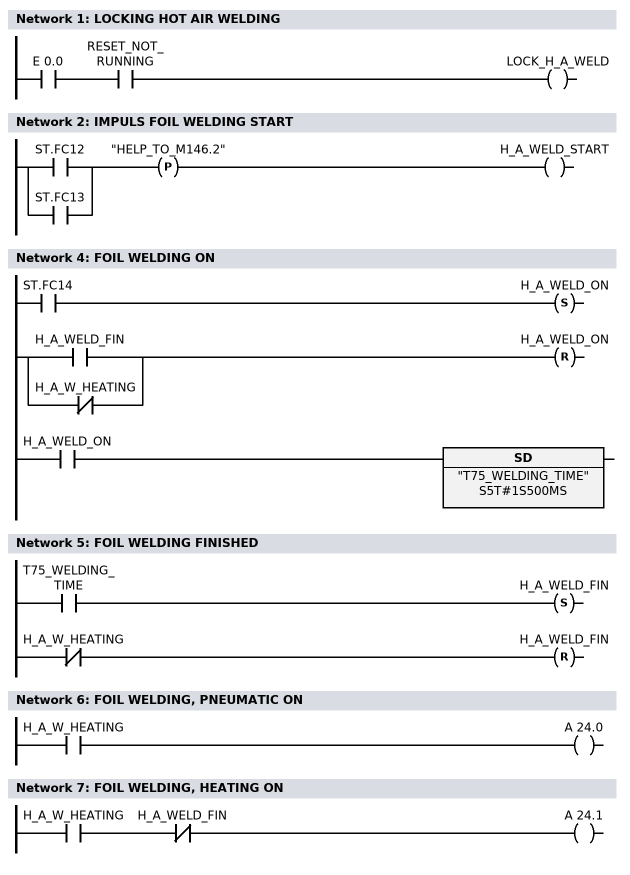
[picture p48: HOT_AIR_WELDING networks 1-7]
NETWORK
TITLE = LOCKING HOT AIR WELDING
//Verriegelung Folie ansiegeln
      A     "E 0.0";
      A     "RESET_NOT_RUNNING";
      =     "LOCK_H_A_WELD";
NETWORK
TITLE = IMPULS FOIL WELDING START 
//Impuls Folie ansiegeln ein
      A(;
      O     "ST.FC12";
      O     "ST.FC13";
      );
      FP    "HELP_TO_M146.2";
      =     "H_A_WELD_START";
NETWORK
TITLE = FOIL WELDING HEATING 
//Folie ansiegeln ein
      A(;
      A     "H_A_WELD_START";
      S     "H_A_W_HEATING";
      A(;
      ON    "LOCK_H_A_WELD";
      O     "T74_HEATING_TIME";
      );
      R     "H_A_W_HEATING";
      A     "H_A_W_HEATING";
      );
      A     "H_A_WELD_FIN";
      L     S5T#15S;
      SD    "T74_HEATING_TIME";
NETWORK
TITLE = FOIL WELDING ON
//Folie ansiegeln aktiv
      A     "ST.FC14";
      S     "H_A_WELD_ON";
      A(;
      O     "H_A_WELD_FIN";
      ON    "H_A_W_HEATING";
      );
      R     "H_A_WELD_ON";
      A     "H_A_WELD_ON";
      L     S5T#1S500MS;
      SD    "T75_WELDING_TIME";
NETWORK
TITLE = FOIL WELDING FINISHED
//Folie ansiegeln fertig
      A     "T75_WELDING_TIME";
      S     "H_A_WELD_FIN";
      AN    "H_A_W_HEATING";
      R     "H_A_WELD_FIN";
      NOP   0;
NETWORK
TITLE = FOIL WELDING, PNEUMATIC ON
//Folie ansiegeln Luft ein
      A     "H_A_W_HEATING";
      =     "A 24.0";
NETWORK
TITLE = FOIL WELDING, HEATING ON
//Folie ansiegeln Heizung ein
      A     "H_A_W_HEATING";
      AN    "H_A_WELD_FIN";
      =     "A 24.1";
END_FUNCTION

FUNCTION "WELDING" : VOID	// FC 29
TITLE = FILM WELDING, OPTION
AUTHOR : LKA
NAME : WELDING
VERSION : 0.1
BEGIN
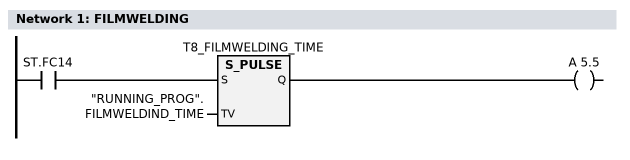
NETWORK
TITLE = FILMWELDING
      A     "ST.FC14";
      L     "RUNNING_PROG".FILMWELDIND_TIME;
      SP    "T8_FILMWELDING_TIME";
      NOP   0;
      NOP   0;
      NOP   0;
      A     "T8_FILMWELDING_TIME";
      =     "A 5.5";
END_FUNCTION

FUNCTION "TURNTABLE_COUNTERS" : VOID	// FC 32
TITLE = TURNTABLE COUNTERS AND TIMERS
//HELP FUNCTION TO PROGRAM, COMMON COUNTERS USED IN WRAPPING PROGRAMMS
AUTHOR : LKA
NAME : FROM_TOP
VERSION : 0.1
BEGIN
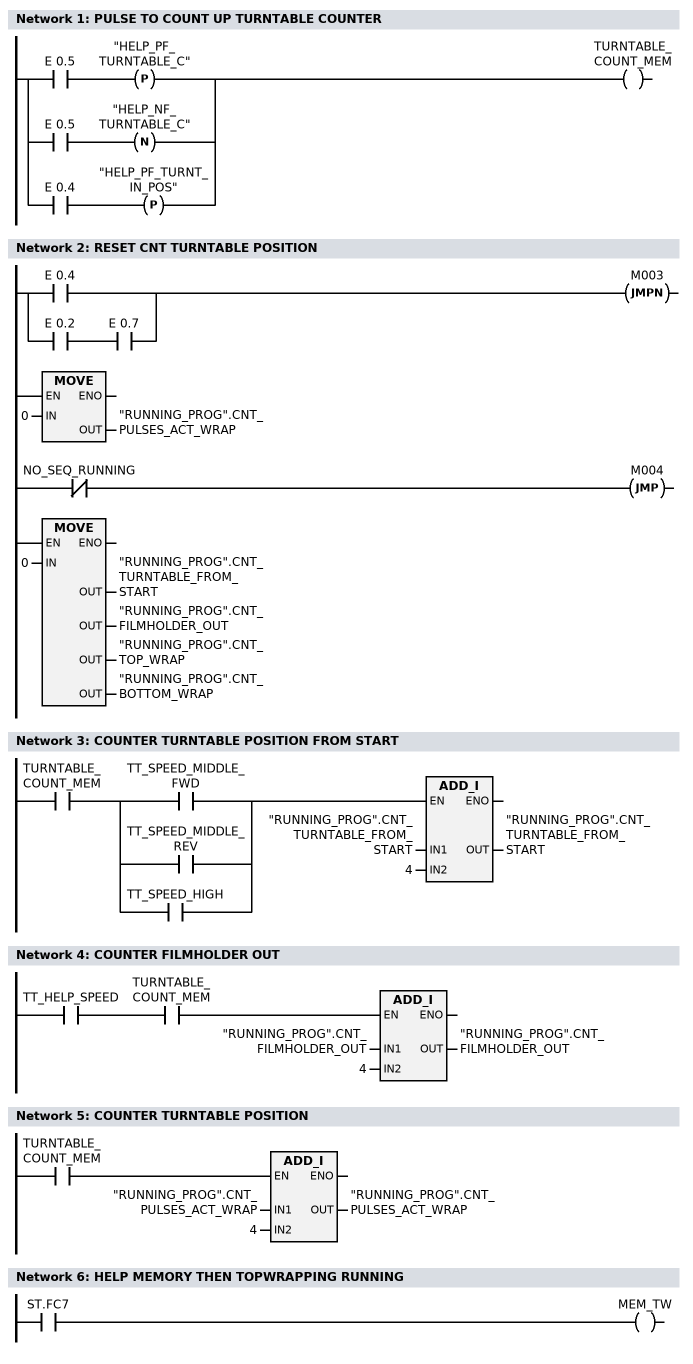
NETWORK
TITLE = PULSE TO COUNT UP TURNTABLE COUNTER
      A     "E 0.5";
      FP    "HELP_PF_TURNTABLE_C";
      O(;
      A     "E 0.5";
      FN    "HELP_NF_TURNTABLE_C";
      );
      O(;
      A     "E 0.4";
      FP    "HELP_PF_TURNT_IN_POS";
      );
      =     "TURNTABLE_COUNT_MEM";
NETWORK
TITLE = RESET CNT TURNTABLE POSITION
//RESETA BORD POSITIONS RÄKNARE
      O     "E 0.4";
      O;
      A     "E 0.2";
      A     "E 0.7";
      JCN   M003;
      L     0;
      T     "RUNNING_PROG".CNT_PULSES_ACT_WRAP;
M003: NOP   0;
      AN    "NO_SEQ_RUNNING";	// OM INTE NÅGON CYKEL KÖRS
      JC    M004;
      L     0;
      T     "RUNNING_PROG".CNT_TURNTABLE_FROM_START;
      T     "RUNNING_PROG".CNT_FILMHOLDER_OUT;
      T     "RUNNING_PROG".CNT_TOP_WRAP;
      T     "RUNNING_PROG".CNT_BOTTOM_WRAP;
M004: NOP   0;
NETWORK
TITLE = COUNTER TURNTABLE POSITION FROM START
//RÄKNARE BORD POSITION
      A     "TURNTABLE_COUNT_MEM";
      A(;
      O     "TT_SPEED_MIDDLE_FWD";
      O     "TT_SPEED_MIDDLE_REV";
      O     "TT_SPEED_HIGH";
      );
      JNB   _008;
      L     "RUNNING_PROG".CNT_TURNTABLE_FROM_START;
      L     4;
      +I;
      T     "RUNNING_PROG".CNT_TURNTABLE_FROM_START;
_008: NOP   0;
NETWORK
TITLE = COUNTER FILMHOLDER OUT
//RÄKNARE FILMHÅLLARARM UT, samt när byte till hög fart skall ske!
      A     "TT_HELP_SPEED";
      A     "TURNTABLE_COUNT_MEM";
      JNB   _00b;
      L     "RUNNING_PROG".CNT_FILMHOLDER_OUT;
      L     4;
      +I;
      T     "RUNNING_PROG".CNT_FILMHOLDER_OUT;
_00b: NOP   0;
NETWORK
TITLE = COUNTER TURNTABLE POSITION
//RÄKNARE BORD POSITION
      A     "TURNTABLE_COUNT_MEM";
      JNB   _010;
      L     "RUNNING_PROG".CNT_PULSES_ACT_WRAP;
      L     4;
      +I;
      T     "RUNNING_PROG".CNT_PULSES_ACT_WRAP;
_010: NOP   0;
NETWORK
TITLE = HELP MEMORY THEN TOPWRAPPING RUNNING
//HJÄLP MINNE FÖR NÄR TOPP VARV KÖRS
      A     "ST.FC7";
      =     "MEM_TW";
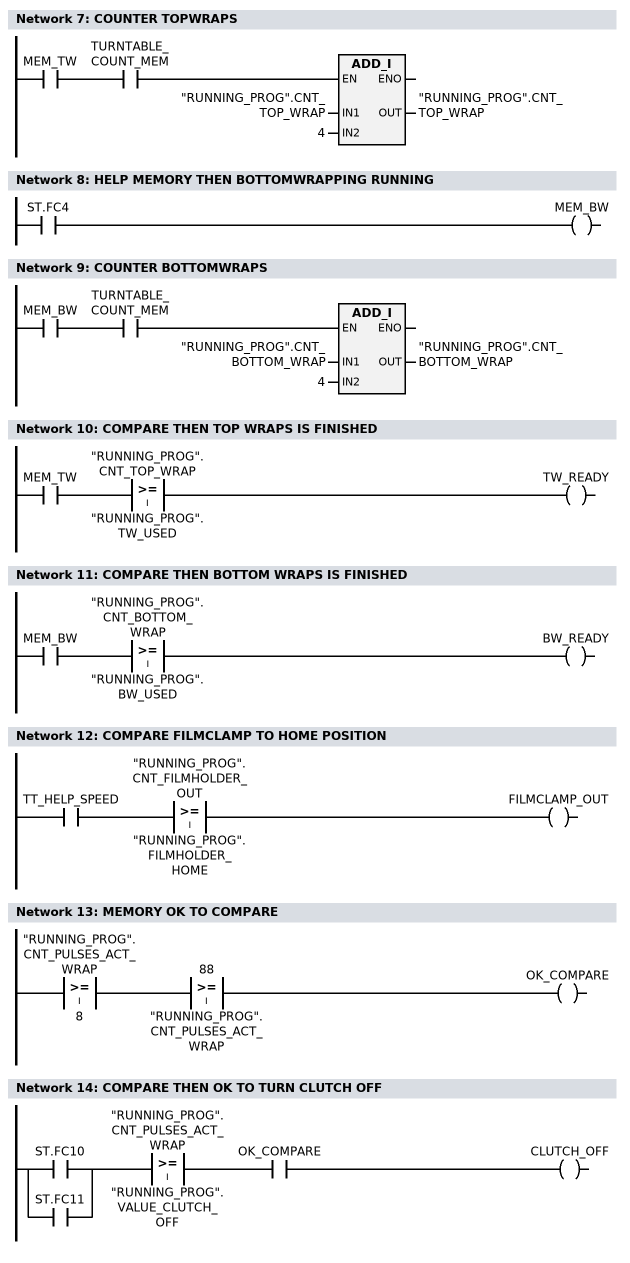
NETWORK
TITLE = COUNTER TOPWRAPS
//RÄKNARE TOPP VARV
      A     "MEM_TW";
      A     "TURNTABLE_COUNT_MEM";
      JNB   _011;
      L     "RUNNING_PROG".CNT_TOP_WRAP;
      L     4;
      +I;
      T     "RUNNING_PROG".CNT_TOP_WRAP;
_011: NOP   0;
NETWORK
TITLE = HELP MEMORY THEN BOTTOMWRAPPING RUNNING
//HJÄLP MINNE FÖR NÄR BOTTEN VARV KÖRS
      A     "ST.FC4";
      =     "MEM_BW";
NETWORK
TITLE = COUNTER BOTTOMWRAPS
//RÄKNARE BOTTEN VARV
      A     "MEM_BW";
      A     "TURNTABLE_COUNT_MEM";
      JNB   _012;
      L     "RUNNING_PROG".CNT_BOTTOM_WRAP;
      L     4;
      +I;
      T     "RUNNING_PROG".CNT_BOTTOM_WRAP;
_012: NOP   0;
NETWORK
TITLE = COMPARE THEN TOP WRAPS IS FINISHED
//HJÄLP MINNE TILL NÄR TOPPVARV ÄR KLARA
      A     "MEM_TW";
      A(;
      L     "RUNNING_PROG".CNT_TOP_WRAP;
      L     "RUNNING_PROG".TW_USED;
      >=I;
      );
      =     "TW_READY";
NETWORK
TITLE = COMPARE THEN BOTTOM WRAPS IS FINISHED
//HJÄLP MINNE TILL NÄR BOTTENVARV ÄR KLARA
//BYTT DB12.DBW80 MOT 78??!!!!
      A     "MEM_BW";
      A(;
      L     "RUNNING_PROG".CNT_BOTTOM_WRAP;
      L     "RUNNING_PROG".BW_USED;
      >=I;
      );
      =     "BW_READY";
NETWORK
TITLE = COMPARE FILMCLAMP TO HOME POSITION
//HJÄLP MINNE TILL NÄR FILMHÅLLARARM SKALL UT
//
      A     "TT_HELP_SPEED";
      A(;
      L     "RUNNING_PROG".CNT_FILMHOLDER_OUT;
      L     "RUNNING_PROG".FILMHOLDER_HOME;
      >=I;
      );
      =     "FILMCLAMP_OUT";
NETWORK
TITLE = MEMORY OK TO COMPARE
      A(;
      L     "RUNNING_PROG".CNT_PULSES_ACT_WRAP;
      L     8;
      >=I;
      );
      A(;
      L     88;
      L     "RUNNING_PROG".CNT_PULSES_ACT_WRAP;
      >=I;
      );
      =     "OK_COMPARE";
NETWORK
TITLE = COMPARE THEN OK TO TURN CLUTCH OFF
      A(;
      O     "ST.FC10";
      O     "ST.FC11";
      );
      A(;
      L     "RUNNING_PROG".CNT_PULSES_ACT_WRAP;
      L     "RUNNING_PROG".VALUE_CLUTCH_OFF;
      >=I;
      );
      A     "OK_COMPARE";
      =     "CLUTCH_OFF";
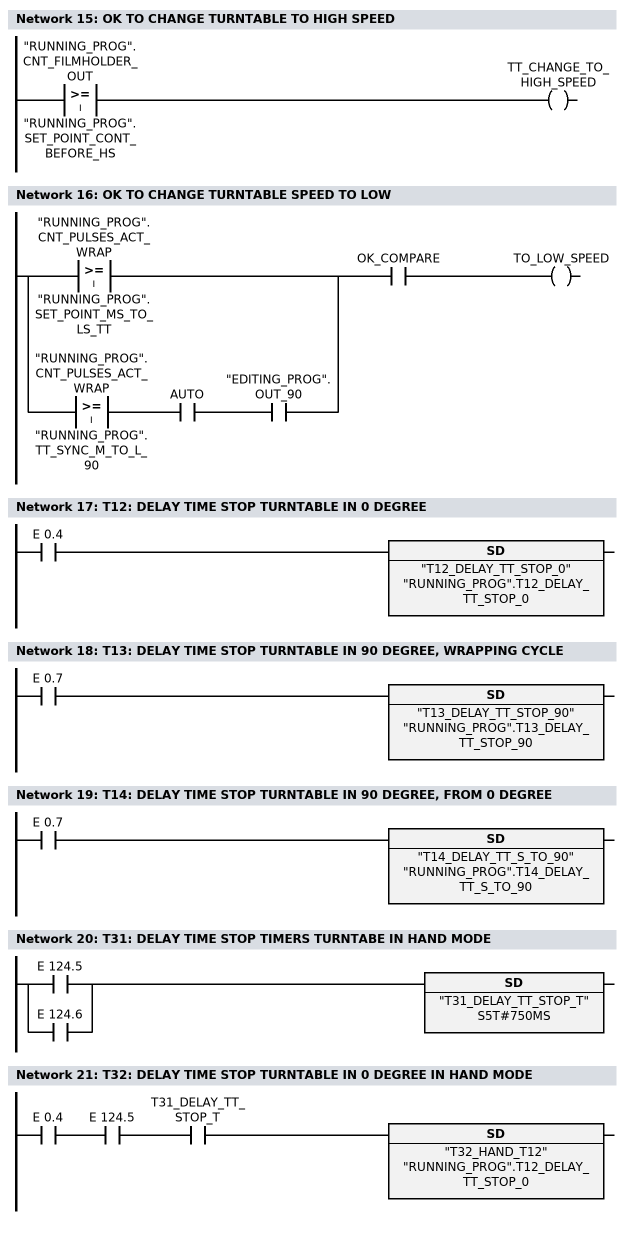
NETWORK
TITLE = OK TO CHANGE TURNTABLE TO HIGH SPEED
//HJÄLP MINNE TILL NÄR BORDET ÄR I POSITION SÅ DET ÄR OK ATT ÖKA TILL HÖGFART
      L     "RUNNING_PROG".CNT_FILMHOLDER_OUT;
      L     "RUNNING_PROG".SET_POINT_CONT_BEFORE_HS;
      >=I;
      =     "TT_CHANGE_TO_HIGH_SPEED";
NETWORK
TITLE = OK TO CHANGE TURNTABLE SPEED TO LOW
      A(;
      O(;
      L     "RUNNING_PROG".CNT_PULSES_ACT_WRAP;
      L     "RUNNING_PROG".SET_POINT_MS_TO_LS_TT;
      >=I;
      );
      O;
      A(;
      L     "RUNNING_PROG".CNT_PULSES_ACT_WRAP;
      L     "RUNNING_PROG".TT_SYNC_M_TO_L_90;
      >=I;
      );
      A     "AUTO";
      A     "EDITING_PROG".OUT_90;
      );
      A     "OK_COMPARE";
      =     "TO_LOW_SPEED";
NETWORK
TITLE = T12: DELAY TIME STOP TURNTABLE IN 0 DEGREE
      A     "E 0.4";
      L     "RUNNING_PROG".T12_DELAY_TT_STOP_0;
      SD    "T12_DELAY_TT_STOP_0";
NETWORK
TITLE = T13: DELAY TIME STOP TURNTABLE IN 90 DEGREE, WRAPPING CYCLE
      A     "E 0.7";
      L     "RUNNING_PROG".T13_DELAY_TT_STOP_90;
      SD    "T13_DELAY_TT_STOP_90";
NETWORK
TITLE = T14: DELAY TIME STOP TURNTABLE IN 90 DEGREE, FROM 0 DEGREE
      A     "E 0.7";
      L     "RUNNING_PROG".T14_DELAY_TT_S_TO_90;
      SD    "T14_DELAY_TT_S_TO_90";
NETWORK
TITLE = T31: DELAY TIME STOP TIMERS TURNTABE IN HAND MODE
      O     "E 124.5";
      O     "E 124.6";
      L     S5T#750MS;
      SD    "T31_DELAY_TT_STOP_T";
NETWORK
TITLE = T32: DELAY TIME STOP TURNTABLE IN 0 DEGREE IN HAND MODE
      A     "E 0.4";
      A     "E 124.5";
      A     "T31_DELAY_TT_STOP_T";
      L     "RUNNING_PROG".T12_DELAY_TT_STOP_0;
      SD    "T32_HAND_T12";
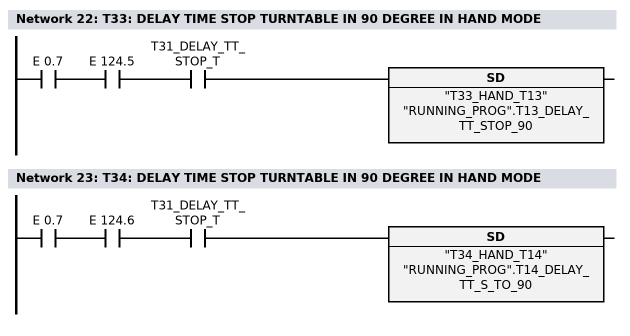
NETWORK
TITLE = T33: DELAY TIME STOP TURNTABLE IN 90 DEGREE IN HAND MODE
      A     "E 0.7";
      A     "E 124.5";
      A     "T31_DELAY_TT_STOP_T";
      L     "RUNNING_PROG".T13_DELAY_TT_STOP_90;
      SD    "T33_HAND_T13";
NETWORK
TITLE = T34: DELAY TIME STOP TURNTABLE IN 90 DEGREE IN HAND MODE
      A     "E 0.7";
      A     "E 124.6";
      A     "T31_DELAY_TT_STOP_T";
      L     "RUNNING_PROG".T14_DELAY_TT_S_TO_90;
      SD    "T34_HAND_T14";
END_FUNCTION

FUNCTION "CARRIAGE_COUNTERS" : VOID	// FC 33
TITLE = CARRIAGE COUNTERS
//HELP FUNCTION TO PROGRAM, COMMON COUNTERS USED IN WRAPPING PROGRAMMS
AUTHOR : LKA
NAME : FROM_TOP
VERSION : 0.1
BEGIN
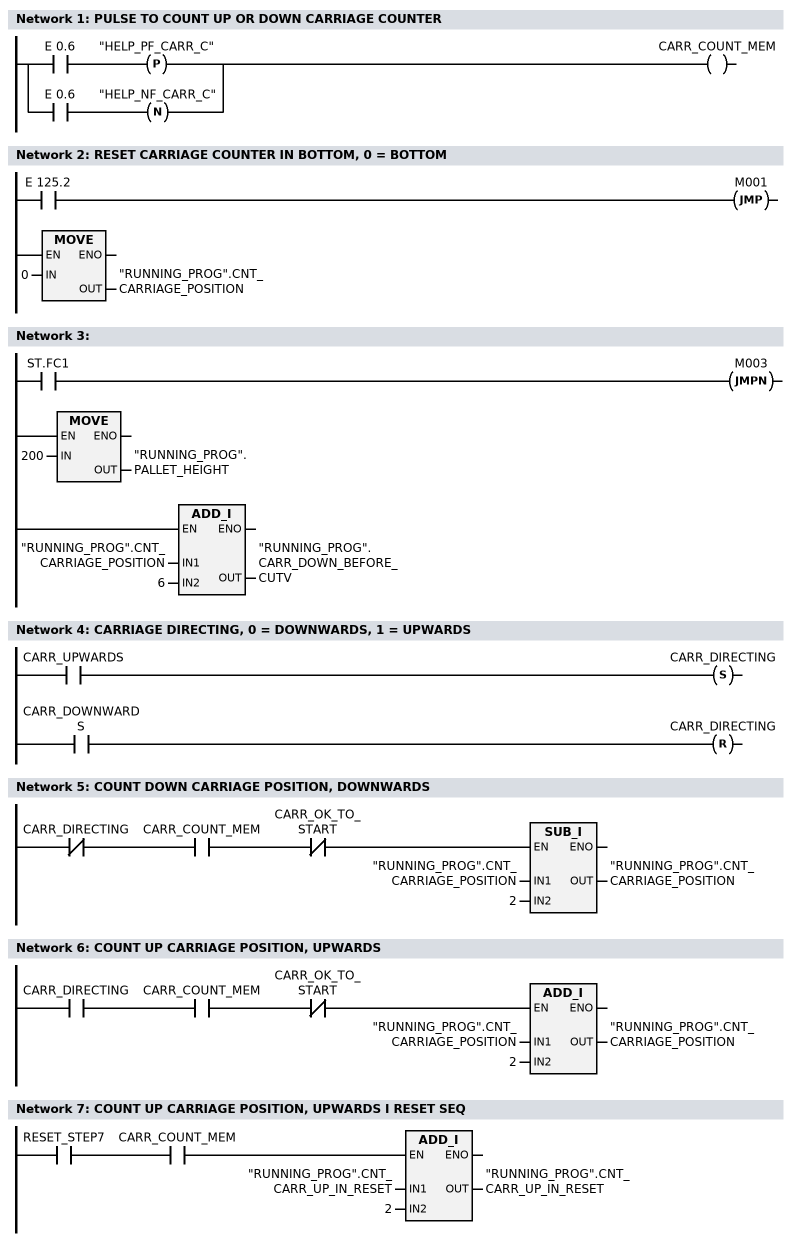
NETWORK
TITLE = PULSE TO COUNT UP OR DOWN CARRIAGE COUNTER
      A     "E 0.6";
      FP    "HELP_PF_CARR_C";
      O(;
      A     "E 0.6";
      FN    "HELP_NF_CARR_C";
      );
      =     "CARR_COUNT_MEM";
NETWORK
TITLE = RESET CARRIAGE COUNTER IN BOTTOM, 0 = BOTTOM
//RESETA HISS POS I BOTTENLÄGET
      A     "E 125.2";
      JC    M001;
      L     0;
      T     "RUNNING_PROG".CNT_CARRIAGE_POSITION;
M001: NOP   0;
NETWORK
TITLE =
      A     "ST.FC1";
      JCN   M003;
      L     200;
      T     "RUNNING_PROG".PALLET_HEIGHT;
      L     "RUNNING_PROG".CNT_CARRIAGE_POSITION;
      L     6;
      +I;
      T     "RUNNING_PROG".CARR_DOWN_BEFORE_CUTV;
M003: NOP   0;
NETWORK
TITLE = CARRIAGE DIRECTING, 0 = DOWNWARDS, 1 = UPWARDS
//HISS RIKTNING, 0 = NEDÅT, 1 = UPPÅT
      A     "CARR_UPWARDS";
      S     "CARR_DIRECTING";
      A     "CARR_DOWNWARDS";
      R     "CARR_DIRECTING";
      NOP   0;
NETWORK
TITLE = COUNT DOWN CARRIAGE POSITION, DOWNWARDS
//RÄKNA NED HISS POS NÄR HISSEN ÅKER NEDÅT
      AN    "CARR_DIRECTING";
      A     "CARR_COUNT_MEM";
      AN    "CARR_OK_TO_START";
      JNB   _00b;
      L     "RUNNING_PROG".CNT_CARRIAGE_POSITION;
      L     2;
      -I;
      T     "RUNNING_PROG".CNT_CARRIAGE_POSITION;
_00b: NOP   0;
NETWORK
TITLE = COUNT UP CARRIAGE POSITION, UPWARDS
//RÄKNA UPP HISS POS NÄR HISSEN ÅKER UPPÅT
      A     "CARR_DIRECTING";
      A     "CARR_COUNT_MEM";
      AN    "CARR_OK_TO_START";
      JNB   _00c;
      L     "RUNNING_PROG".CNT_CARRIAGE_POSITION;
      L     2;
      +I;
      T     "RUNNING_PROG".CNT_CARRIAGE_POSITION;
_00c: NOP   0;
NETWORK
TITLE = COUNT UP CARRIAGE POSITION, UPWARDS I RESET SEQ
//RÄKNA UPP HISS POS NÄR HISSEN ÅKER UPPÅT
      A     "RESET_STEP7";
      A     "CARR_COUNT_MEM";
      JNB   _00d;
      L     "RUNNING_PROG".CNT_CARR_UP_IN_RESET;
      L     2;
      +I;
      T     "RUNNING_PROG".CNT_CARR_UP_IN_RESET;
_00d: NOP   0;
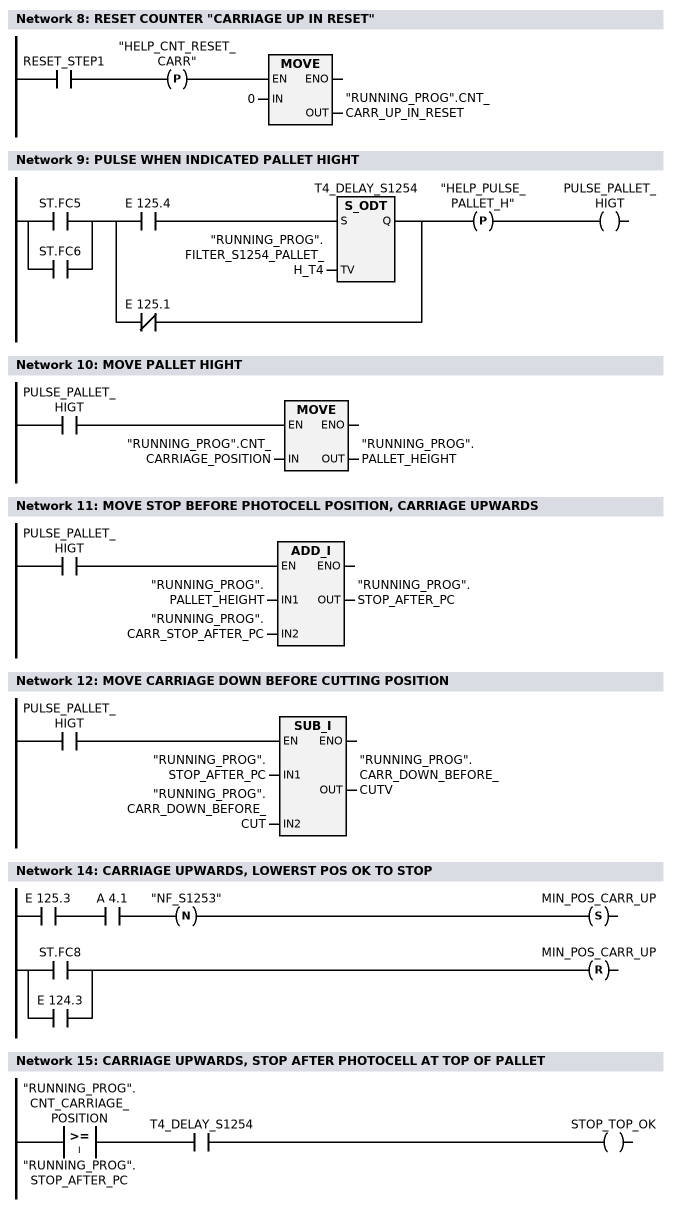
NETWORK
TITLE = RESET COUNTER "CARRIAGE UP IN RESET"
      A     "RESET_STEP1";
      FP    "HELP_CNT_RESET_CARR";
      JNB   _00e;
      L     0;
      T     "RUNNING_PROG".CNT_CARR_UP_IN_RESET;
_00e: NOP   0;
NETWORK
TITLE = PULSE WHEN INDICATED PALLET HIGHT
//SÄTTER PALL HÖJD
//TILLSLAGSTIMMER = FILTER
      A(;
      O     "ST.FC5";
      O     "ST.FC6";
      );
      A(;
      O(;
      A     "E 125.4";
      L     "RUNNING_PROG".FILTER_S1254_PALLET_H_T4;
      SD    "T4_DELAY_S1254";
      NOP   0;
      NOP   0;
      NOP   0;
      A     "T4_DELAY_S1254";
      );
      ON    "E 125.1";
      );
      FP    "HELP_PULSE_PALLET_H";
      =     "PULSE_PALLET_HIGT";
NETWORK
TITLE = MOVE PALLET HIGHT
//SÄTTER PALL HÖJD
      A     "PULSE_PALLET_HIGT";
      JNB   _00f;
      L     "RUNNING_PROG".CNT_CARRIAGE_POSITION;
      T     "RUNNING_PROG".PALLET_HEIGHT;
_00f: NOP   0;
NETWORK
TITLE = MOVE STOP BEFORE PHOTOCELL POSITION, CARRIAGE UPWARDS
      A     "PULSE_PALLET_HIGT";
      JNB   _010;
      L     "RUNNING_PROG".PALLET_HEIGHT;
      L     "RUNNING_PROG".CARR_STOP_AFTER_PC;
      +I;
      T     "RUNNING_PROG".STOP_AFTER_PC;
_010: NOP   0;
NETWORK
TITLE = MOVE CARRIAGE DOWN BEFORE CUTTING POSITION
      A     "PULSE_PALLET_HIGT";
      JNB   _011;
      L     "RUNNING_PROG".STOP_AFTER_PC;
      L     "RUNNING_PROG".CARR_DOWN_BEFORE_CUT;
      -I;
      T     "RUNNING_PROG".CARR_DOWN_BEFORE_CUTV;
_011: NOP   0;
NETWORK
TITLE =
      A     "PULSE_PALLET_HIGT";
      JCN   M004;
      L     "RUNNING_PROG".CARR_DOWN_BEFORE_CUTV;
      L     "RUNNING_PROG".LOWERST_OK_CUT;
      >I;
      JC    M005;
      T     "RUNNING_PROG".CARR_DOWN_BEFORE_CUTV;
M005: NOP   0;
      L     "RUNNING_PROG".STOP_AFTER_PC;
      L     "RUNNING_PROG".LOWERST_OK_CUT;
      >I;
      JC    M004;
      T     "RUNNING_PROG".STOP_AFTER_PC;
M004: NOP   0;
NETWORK
TITLE = CARRIAGE UPWARDS, LOWERST POS OK TO STOP
      A     "E 125.3";
      A     "A 4.1";
      FN    "NF_S1253";
      S     "MIN_POS_CARR_UP";
      A(;
      O     "ST.FC8";
      O     "E 124.3";
      );
      R     "MIN_POS_CARR_UP";
      NOP   0;
NETWORK
TITLE = CARRIAGE UPWARDS, STOP AFTER PHOTOCELL AT TOP OF PALLET
//HJÄLP MINNE TILL NÄR HISSEN STANNAR I TOPP AV PALL, FILMNING AV PALL
      A(;
      L     "RUNNING_PROG".CNT_CARRIAGE_POSITION;
      L     "RUNNING_PROG".STOP_AFTER_PC;
      >=I;
      );
      A     "T4_DELAY_S1254";
      =     "STOP_TOP_OK";
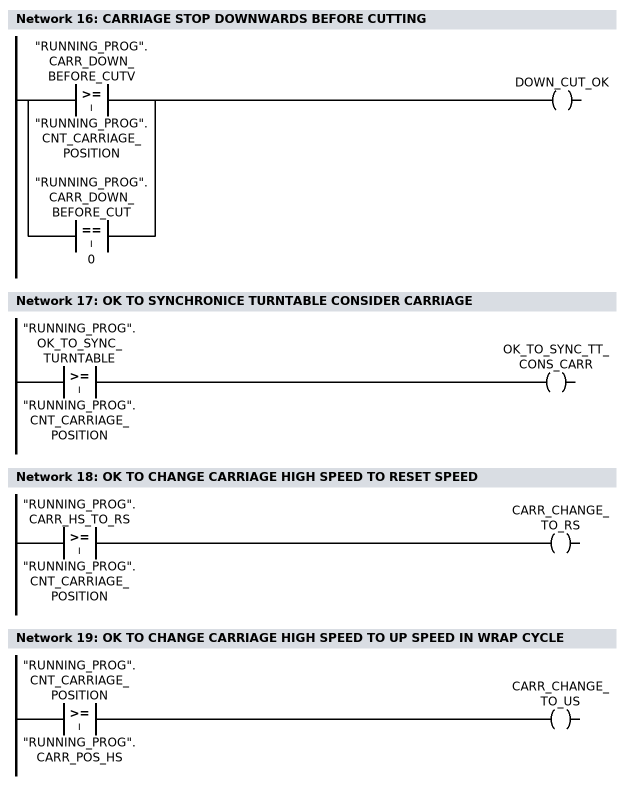
NETWORK
TITLE = CARRIAGE STOP DOWNWARDS BEFORE CUTTING
//HJÄLP MINNE TILL NÄR HISSEN STANNAR PÅ VÄG NED FÖRE AVSKÄRNING AV FILM
      O(;
      L     "RUNNING_PROG".CARR_DOWN_BEFORE_CUTV;
      L     "RUNNING_PROG".CNT_CARRIAGE_POSITION;
      >=I;
      );
      O(;
      L     "RUNNING_PROG".CARR_DOWN_BEFORE_CUT;
      L     0;
      ==I;
      );
      =     "DOWN_CUT_OK";
NETWORK
TITLE = OK TO SYNCHRONICE TURNTABLE CONSIDER CARRIAGE
//HJÄLP MINNE TILL NÄR HISSEN ÄR I POSITION SÅ DET ÄR OK ATT BÖRJA SYNKRONICERA 
//BORDET.
      L     "RUNNING_PROG".OK_TO_SYNC_TURNTABLE;
      L     "RUNNING_PROG".CNT_CARRIAGE_POSITION;
      >=I;
      =     "OK_TO_SYNC_TT_CONS_CARR";
NETWORK
TITLE = OK TO CHANGE CARRIAGE HIGH SPEED TO RESET SPEED
      L     "RUNNING_PROG".CARR_HS_TO_RS;
      L     "RUNNING_PROG".CNT_CARRIAGE_POSITION;
      >=I;
      =     "CARR_CHANGE_TO_RS";
NETWORK
TITLE = OK TO CHANGE CARRIAGE HIGH SPEED TO UP SPEED IN WRAP CYCLE
      L     "RUNNING_PROG".CNT_CARRIAGE_POSITION;
      L     "RUNNING_PROG".CARR_POS_HS;
      >=I;
      =     "CARR_CHANGE_TO_US";
END_FUNCTION

FUNCTION "COUNTERS" : VOID	// FC 34
TITLE = COUNTERS
AUTHOR : LKA
NAME : FROM_TOP
VERSION : 0.1
BEGIN
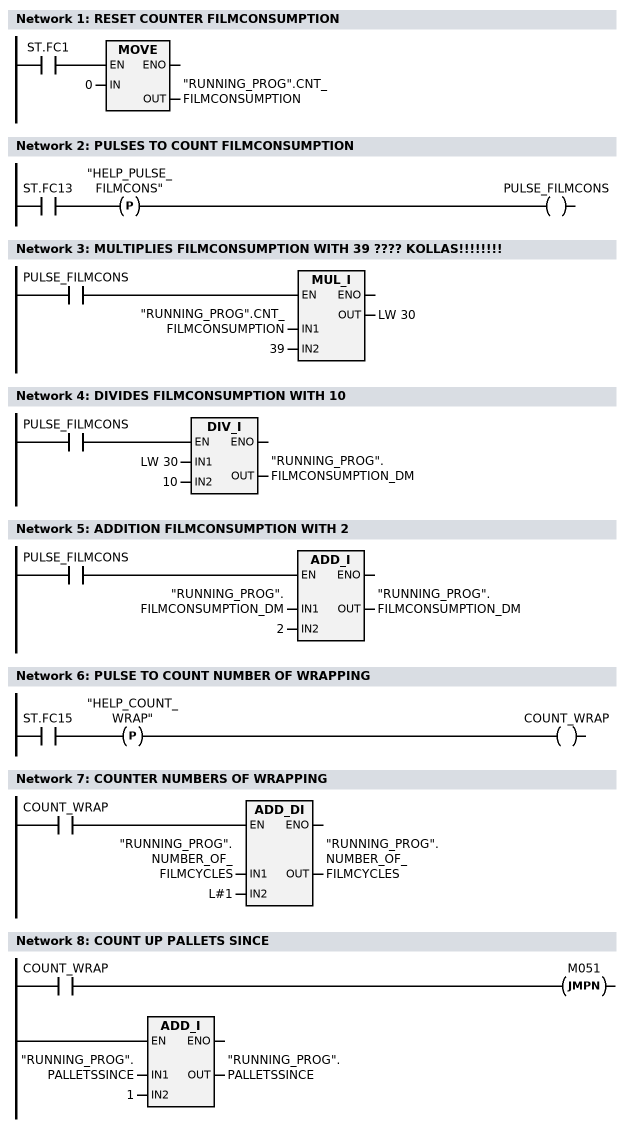
NETWORK
TITLE = RESET COUNTER FILMCONSUMPTION
      A     "ST.FC1";
      JNB   _003;
      L     0;
      T     "RUNNING_PROG".CNT_FILMCONSUMPTION;
_003: NOP   0;
NETWORK
TITLE = PULSES TO COUNT FILMCONSUMPTION
      A     "ST.FC13";
      FP    "HELP_PULSE_FILMCONS";
      =     "PULSE_FILMCONS";
NETWORK
TITLE = MULTIPLIES FILMCONSUMPTION WITH 39 ???? KOLLAS!!!!!!!!
      A     "PULSE_FILMCONS";
      JNB   _007;
      L     "RUNNING_PROG".CNT_FILMCONSUMPTION;
      L     39;
      *I;
      T     LW 30;
_007: NOP   0;
NETWORK
TITLE = DIVIDES FILMCONSUMPTION WITH 10
      A     "PULSE_FILMCONS";
      JNB   _013;
      L     LW 30;
      L     10;
      /I;
      T     "RUNNING_PROG".FILMCONSUMPTION_DM;
_013: NOP   0;
NETWORK
TITLE = ADDITION FILMCONSUMPTION WITH 2
      A     "PULSE_FILMCONS";
      JNB   _017;
      L     "RUNNING_PROG".FILMCONSUMPTION_DM;
      L     2;
      +I;
      T     "RUNNING_PROG".FILMCONSUMPTION_DM;
_017: NOP   0;
NETWORK
TITLE = PULSE TO COUNT NUMBER OF WRAPPING
//PULS TILL RÄKNARE FILMCYKLER
      A     "ST.FC15";
      FP    "HELP_COUNT_WRAP";
      =     "COUNT_WRAP";
NETWORK
TITLE = COUNTER NUMBERS OF WRAPPING
//RÄKNARE FILMCYKLER
      A     "COUNT_WRAP";
      JNB   _01b;
      L     "RUNNING_PROG".NUMBER_OF_FILMCYCLES;
      L     L#1;
      +D;
      T     "RUNNING_PROG".NUMBER_OF_FILMCYCLES;
_01b: NOP   0;
NETWORK
TITLE = COUNT UP PALLETS SINCE
      A     "COUNT_WRAP";
      JCN   M051;
      L     "RUNNING_PROG".PALLETSSINCE;
      L     1;
      +I;
      T     "RUNNING_PROG".PALLETSSINCE;
M051: NOP   0;
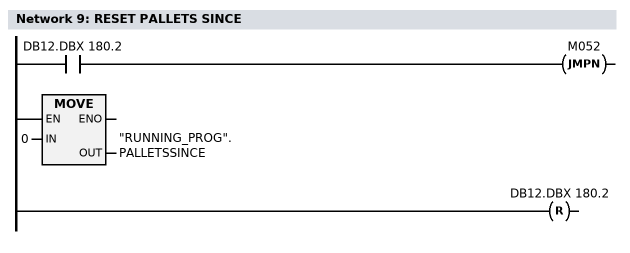
NETWORK
TITLE = RESET PALLETS SINCE
      A     DB12.DBX 180.2;
      JCN   M052;
      L     0;
      T     "RUNNING_PROG".PALLETSSINCE;
      R     DB12.DBX 180.2;
M052: NOP   0;
END_FUNCTION

FUNCTION "CONVEYOR_1" : VOID	// FC 71
VERSION : 0.1
BEGIN
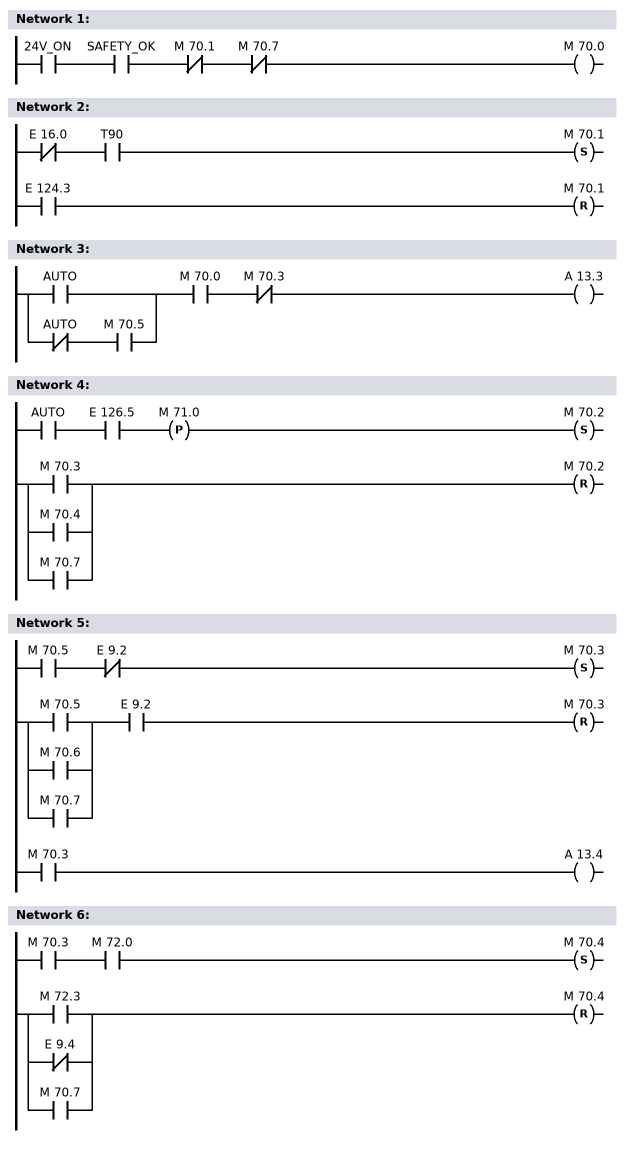
NETWORK
TITLE =
      A     "24V_ON";
      A     "SAFETY_OK";
      AN    "M 70.1";
      AN    "M 70.7";
      =     "M 70.0";
NETWORK
TITLE =
      AN    "E 16.0";
      A     "T90";
      S     "M 70.1";
      A     "E 124.3";
      R     "M 70.1";
      NOP   0;
NETWORK
TITLE =
      A(;
      O     "AUTO";
      O;
      AN    "AUTO";
      A     "M 70.5";
      );
      A     "M 70.0";
      AN    "M 70.3";
      =     "A 13.3";
NETWORK
TITLE =
      A     "AUTO";
      A     "E 126.5";
      FP    M 71.0;
      S     "M 70.2";
      A(;
      O     "M 70.3";
      O     "M 70.4";
      O     "M 70.7";
      );
      R     "M 70.2";
      NOP   0;
NETWORK
TITLE =
      A     "M 70.5";
      AN    "E 9.2";
      S     "M 70.3";
      A(;
      O     "M 70.5";
      O     "M 70.6";
      O     "M 70.7";
      );
      A     "E 9.2";
      R     "M 70.3";
      A     "M 70.3";
      =     "A 13.4";
NETWORK
TITLE =
      A     "M 70.3";
      A     "M 72.0";
      S     "M 70.4";
      A(;
      O     "M 72.3";
      ON    "E 9.4";
      O     "M 70.7";
      );
      R     "M 70.4";
      NOP   0;
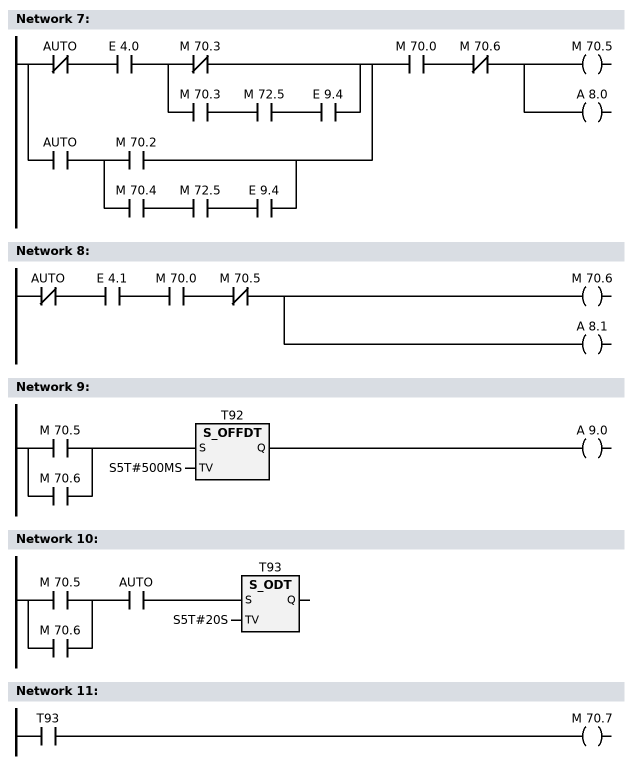
NETWORK
TITLE =
      A(;
      AN    "AUTO";
      A     "E 4.0";
      A(;
      ON    "M 70.3";
      O;
      A     "M 70.3";
      A     "M 72.5";
      A     "E 9.4";
      );
      O;
      A     "AUTO";
      A(;
      O     "M 70.2";
      O;
      A     "M 70.4";
      A     "M 72.5";
      A     "E 9.4";
      );
      );
      A     "M 70.0";
      AN    "M 70.6";
      =     "M 70.5";
      =     "A 8.0";
NETWORK
TITLE =
      AN    "AUTO";
      A     "E 4.1";
      A     "M 70.0";
      AN    "M 70.5";
      =     "M 70.6";
      =     "A 8.1";
NETWORK
TITLE =
      A(;
      O     "M 70.5";
      O     "M 70.6";
      );
      L     S5T#500MS;
      SF    "T92";
      NOP   0;
      NOP   0;
      NOP   0;
      A     "T92";
      =     "A 9.0";
NETWORK
TITLE =
      A(;
      O     "M 70.5";
      O     "M 70.6";
      );
      A     "AUTO";
      L     S5T#20S;
      SD    "T93";
      NOP   0;
      NOP   0;
      NOP   0;
      NOP   0;
NETWORK
TITLE =
      A     "T93";
      =     "M 70.7";
END_FUNCTION

FUNCTION "CONVEYOR_2" : VOID	// FC 72
VERSION : 0.1
BEGIN
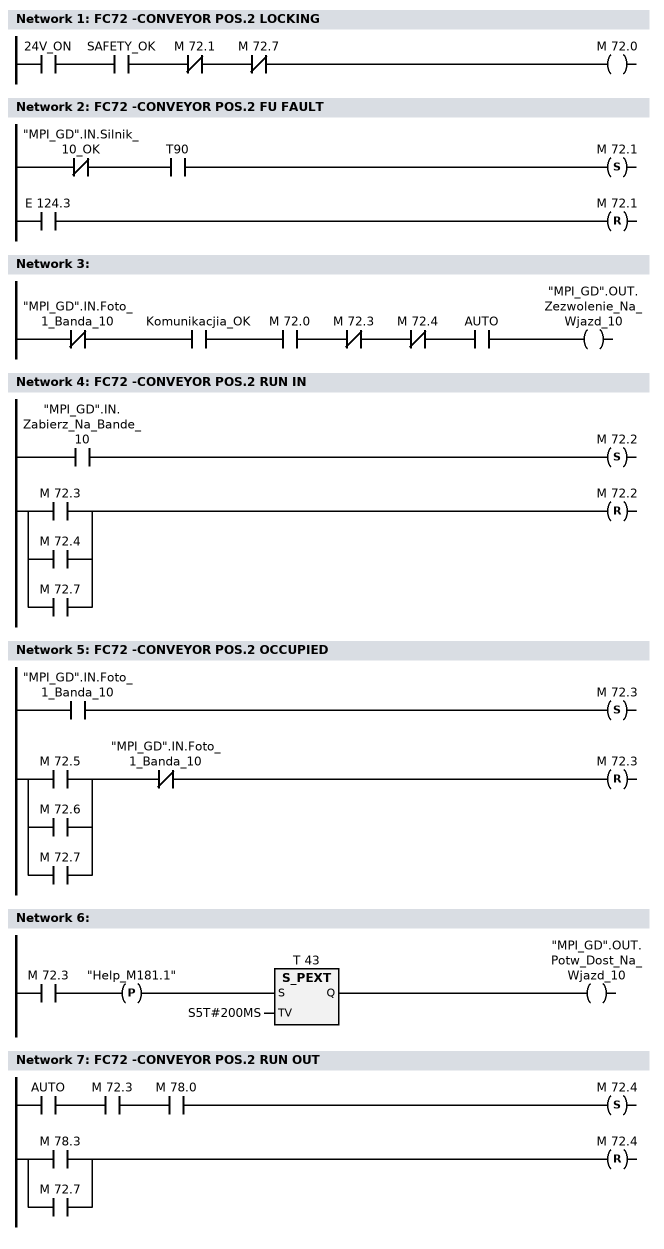
NETWORK
TITLE = FC72 -CONVEYOR POS.2 LOCKING
//Ustawienie obrotnicy na pozycji 0 stopni
      A     "24V_ON";
      A     "SAFETY_OK";
      AN    "M 72.1";
      AN    "M 72.7";
      =     "M 72.0";
NETWORK
TITLE = FC72 -CONVEYOR POS.2 FU FAULT
//Silnik przenosnika jest OK
      AN    "MPI_GD".IN.Silnik_10_OK;
      A     "T90";
      S     "M 72.1";
      A     "E 124.3";
      R     "M 72.1";
      NOP   0;
NETWORK
TITLE =
//Zezwolenie do bandy 9 (szafa)
      AN    "MPI_GD".IN.Foto_1_Banda_10;
      A     "Komunikacjia_OK";
      A     "M 72.0";
      AN    "M 72.3";
      AN    "M 72.4";
      A     "AUTO";
      =     "MPI_GD".OUT.Zezwolenie_Na_Wjazd_10;
NETWORK
TITLE = FC72 -CONVEYOR POS.2 RUN IN
//Wjazd palet na bande
      A     "MPI_GD".IN.Zabierz_Na_Bande_10;
      S     "M 72.2";
      A(;
      O     "M 72.3";
      O     "M 72.4";
      O     "M 72.7";
      );
      R     "M 72.2";
      NOP   0;
NETWORK
TITLE = FC72 -CONVEYOR POS.2 OCCUPIED
//Paleta na przenosniku nr 2 
      A     "MPI_GD".IN.Foto_1_Banda_10;
      S     "M 72.3";
      A(;
      O     "M 72.5";
      O     "M 72.6";
      O     "M 72.7";
      );
      AN    "MPI_GD".IN.Foto_1_Banda_10;
      R     "M 72.3";
      NOP   0;
NETWORK
TITLE =
//Paleta zostala dostarczona
//
      A     "M 72.3";
      FP    "Help_M181.1";
      L     S5T#200MS;
      SE    T 43;
      NOP   0;
      NOP   0;
      NOP   0;
      A     T 43;
      =     "MPI_GD".OUT.Potw_Dost_Na_Wjazd_10;
NETWORK
TITLE = FC72 -CONVEYOR POS.2 RUN OUT
      A     "AUTO";
      A     "M 72.3";
      A     "M 78.0";
      S     "M 72.4";
      A(;
      O     "M 78.3";
      O     "M 72.7";
      );
      R     "M 72.4";
      NOP   0;
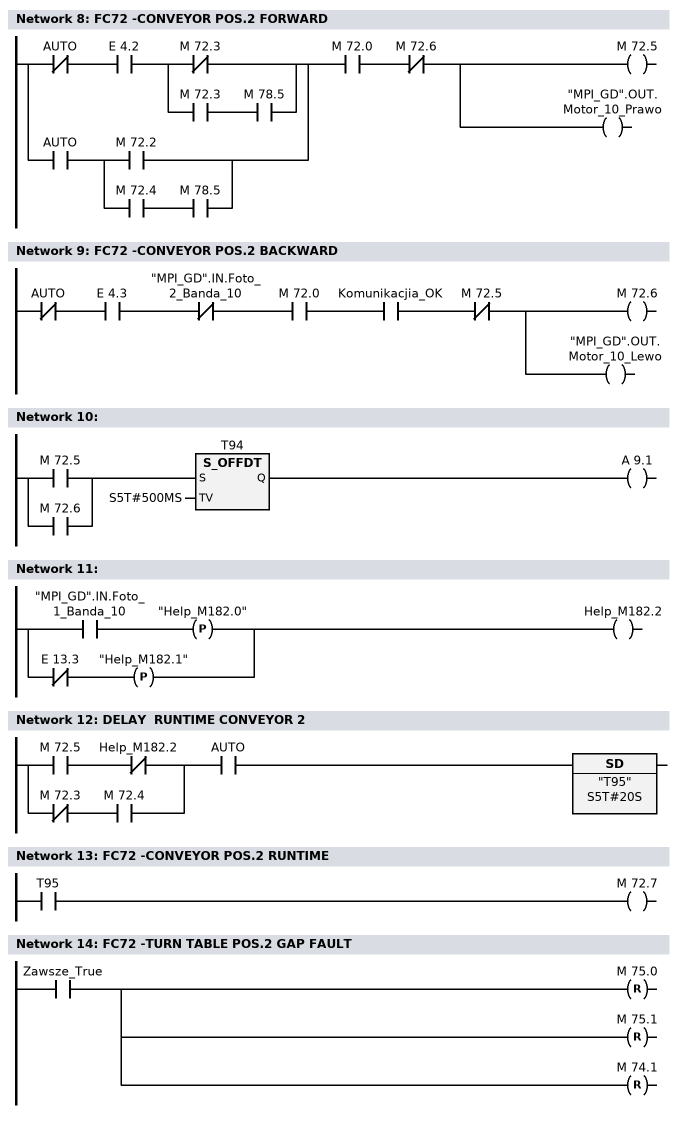
NETWORK
TITLE = FC72 -CONVEYOR POS.2 FORWARD
//Q8.2. Przenosnik jedzie do przodu
      A(;
      AN    "AUTO";
      A     "E 4.2";
      A(;
      ON    "M 72.3";
      O;
      A     "M 72.3";
      A     "M 78.5";
      );
      O;
      A     "AUTO";
      A(;
      O     "M 72.2";
      O;
      A     "M 72.4";
      A     "M 78.5";
      );
      );
      A     "M 72.0";
      AN    "M 72.6";
      =     "M 72.5";
      =     "MPI_GD".OUT.Motor_10_Prawo;
NETWORK
TITLE = FC72 -CONVEYOR POS.2 BACKWARD
//Q8.3 przenosnik jedzie do tylu
      AN    "AUTO";
      A     "E 4.3";
      AN    "MPI_GD".IN.Foto_2_Banda_10;
      A     "M 72.0";
      A     "Komunikacjia_OK";
      AN    "M 72.5";
      =     "M 72.6";
      =     "MPI_GD".OUT.Motor_10_Lewo;
NETWORK
TITLE =
      A(;
      O     "M 72.5";
      O     "M 72.6";
      );
      L     S5T#500MS;
      SF    "T94";
      NOP   0;
      NOP   0;
      NOP   0;
      A     "T94";
      =     "A 9.1";
NETWORK
TITLE =
//Rozlaczenie uplywajacego timera
      A     "MPI_GD".IN.Foto_1_Banda_10;
      FP    "Help_M182.0";
      O(;
      AN    "E 13.3";
      FP    "Help_M182.1";
      );
      =     "Help_M182.2";
NETWORK
TITLE = DELAY  RUNTIME CONVEYOR 2
      A(;
      A     "M 72.5";
      AN    "Help_M182.2";
      O;
      AN    "M 72.3";
      A     "M 72.4";
      );
      A     "AUTO";
      L     S5T#20S;
      SD    "T95";
NETWORK
TITLE = FC72 -CONVEYOR POS.2 RUNTIME
      A     "T95";
      =     "M 72.7";
NETWORK
TITLE = FC72 -TURN TABLE POS.2 GAP FAULT
      A     "Zawsze_True";
      R     "M 75.0";
      R     "M 75.1";
      R     "M 74.1";
END_FUNCTION

FUNCTION "CONVEYOR_3" : VOID	// FC 73
VERSION : 0.1
BEGIN
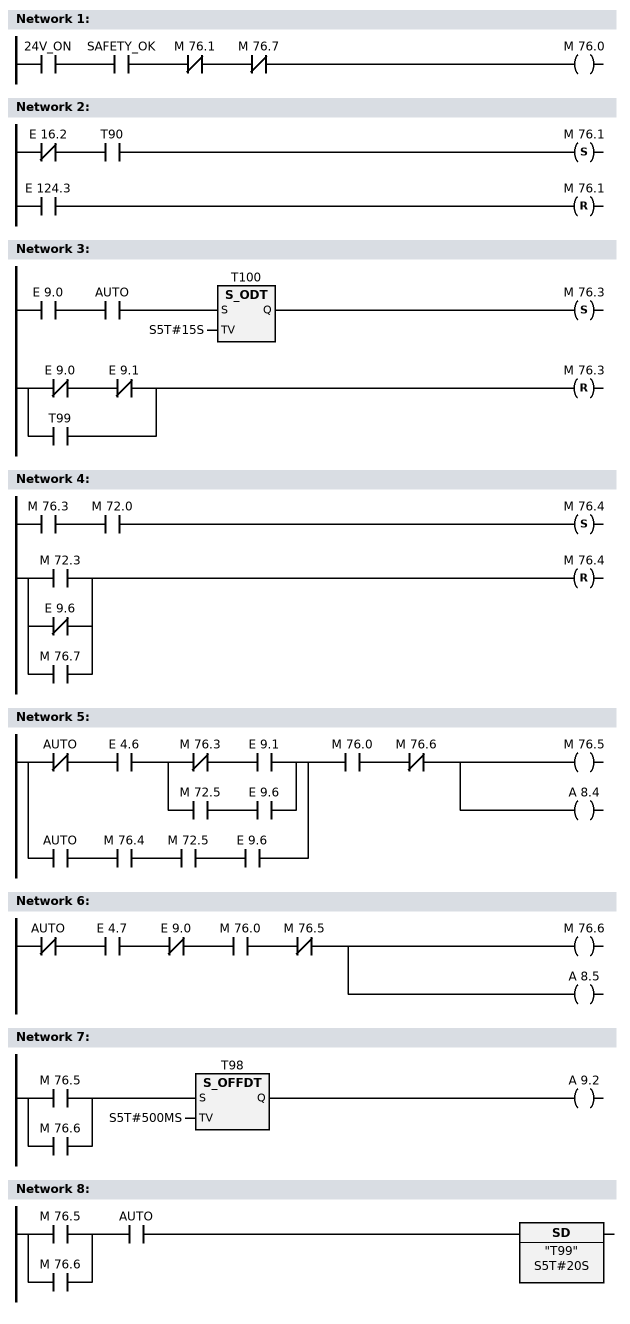
NETWORK
TITLE =
      A     "24V_ON";
      A     "SAFETY_OK";
      AN    "M 76.1";
      AN    "M 76.7";
      =     "M 76.0";
NETWORK
TITLE =
      AN    "E 16.2";
      A     "T90";
      S     "M 76.1";
      A     "E 124.3";
      R     "M 76.1";
      NOP   0;
NETWORK
TITLE =
      A(;
      A     "E 9.0";
      A     "AUTO";
      L     S5T#15S;
      SD    "T100";
      NOP   0;
      NOP   0;
      NOP   0;
      A     "T100";
      );
      S     "M 76.3";
      A(;
      AN    "E 9.0";
      AN    "E 9.1";
      O     "T99";
      );
      R     "M 76.3";
      NOP   0;
NETWORK
TITLE =
      A     "M 76.3";
      A     "M 72.0";
      S     "M 76.4";
      A(;
      O     "M 72.3";
      ON    "E 9.6";
      O     "M 76.7";
      );
      R     "M 76.4";
      NOP   0;
NETWORK
TITLE =
      A(;
      AN    "AUTO";
      A     "E 4.6";
      A(;
      AN    "M 76.3";
      A     "E 9.1";
      O;
      A     "M 72.5";
      A     "E 9.6";
      );
      O;
      A     "AUTO";
      A     "M 76.4";
      A     "M 72.5";
      A     "E 9.6";
      );
      A     "M 76.0";
      AN    "M 76.6";
      =     "M 76.5";
      =     "A 8.4";
NETWORK
TITLE =
      AN    "AUTO";
      A     "E 4.7";
      AN    "E 9.0";
      A     "M 76.0";
      AN    "M 76.5";
      =     "M 76.6";
      =     "A 8.5";
NETWORK
TITLE =
      A(;
      O     "M 76.5";
      O     "M 76.6";
      );
      L     S5T#500MS;
      SF    "T98";
      NOP   0;
      NOP   0;
      NOP   0;
      A     "T98";
      =     "A 9.2";
NETWORK
TITLE =
      A(;
      O     "M 76.5";
      O     "M 76.6";
      );
      A     "AUTO";
      L     S5T#20S;
      SD    "T99";
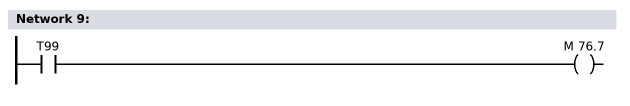
NETWORK
TITLE =
      A     "T99";
      =     "M 76.7";
END_FUNCTION

FUNCTION "CONVEYOR_4" : VOID	// FC 74
TITLE = CONVEYOR POS.4
//
//Bits for conveyor control:
//Bit 0 = Locking conveyor
//Bit 1 = Spare
//Bit 2 = Run in
//Bit 3 = Occupied
//Bit 4 = Run out
//Bit 5 = Forward
//Bit 6 = Backward
//Bit 7 = Runtime
VERSION : 0.1
BEGIN
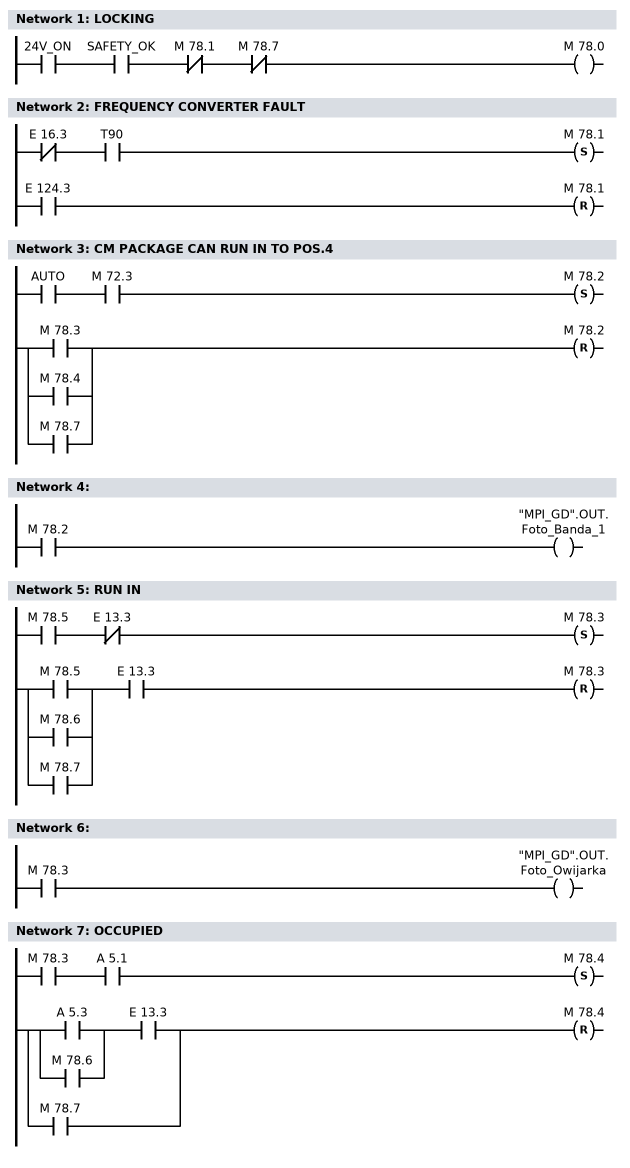
NETWORK
TITLE = LOCKING
      A     "24V_ON";
      A     "SAFETY_OK";
      AN    "M 78.1";
      AN    "M 78.7";
      =     "M 78.0";
NETWORK
TITLE = FREQUENCY CONVERTER FAULT
      AN    "E 16.3";
      A     "T90";
      S     "M 78.1";
      A     "E 124.3";
      R     "M 78.1";
      NOP   0;
NETWORK
TITLE = CM PACKAGE CAN RUN IN TO POS.4
      A     "AUTO";
      A     "M 72.3";
      S     "M 78.2";
      A(;
      O     "M 78.3";
      O     "M 78.4";
      O     "M 78.7";
      );
      R     "M 78.2";
      NOP   0;
NETWORK
TITLE =
      A     "M 78.2";
      =     "MPI_GD".OUT.Foto_Banda_1;
NETWORK
TITLE = RUN IN
      A     "M 78.5";
      AN    "E 13.3";
      S     "M 78.3";
      A(;
      O     "M 78.5";
      O     "M 78.6";
      O     "M 78.7";
      );
      A     "E 13.3";
      R     "M 78.3";
      NOP   0;
NETWORK
TITLE =
      A     "M 78.3";
      =     "MPI_GD".OUT.Foto_Owijarka;
NETWORK
TITLE = OCCUPIED
      A     "M 78.3";
      A     "A 5.1";
      S     "M 78.4";
      A(;
      A(;
      O     "A 5.3";
      O     "M 78.6";
      );
      A     "E 13.3";
      O     "M 78.7";
      );
      R     "M 78.4";
      NOP   0;
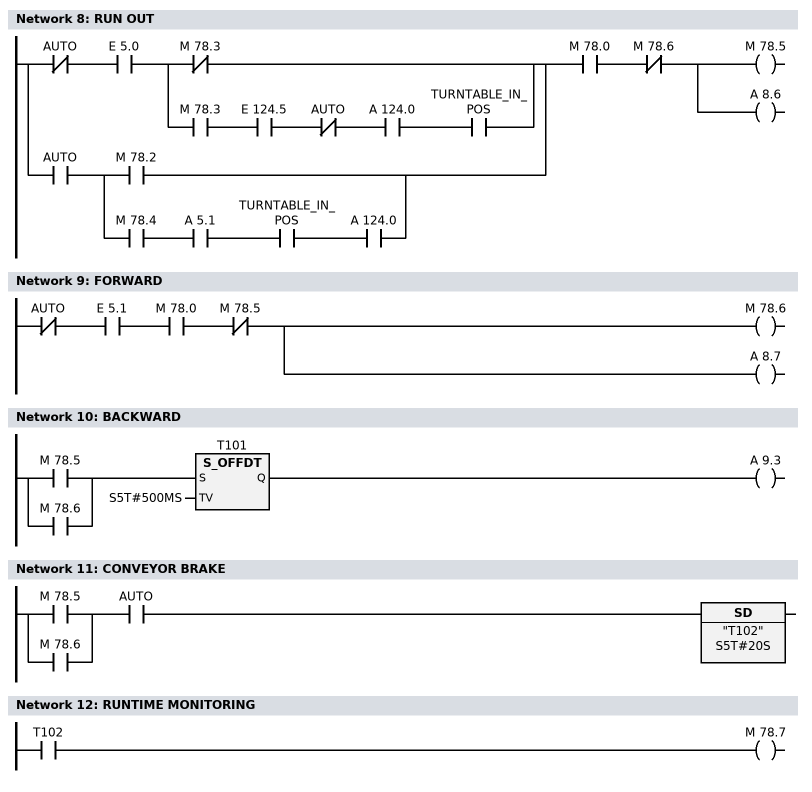
NETWORK
TITLE = RUN OUT
      A(;
      AN    "AUTO";
      A     "E 5.0";
      A(;
      ON    "M 78.3";
      O;
      A     "M 78.3";
      A     "E 124.5";
      AN    "AUTO";
      A     "A 124.0";
      A     "TURNTABLE_IN_POS";
      );
      O;
      A     "AUTO";
      A(;
      O     "M 78.2";
      O;
      A     "M 78.4";
      A     "A 5.1";
      A     "TURNTABLE_IN_POS";
      A     "A 124.0";
      );
      );
      A     "M 78.0";
      AN    "M 78.6";
      =     "M 78.5";
      =     "A 8.6";
NETWORK
TITLE = FORWARD
      AN    "AUTO";
      A     "E 5.1";
      A     "M 78.0";
      AN    "M 78.5";
      =     "M 78.6";
      =     "A 8.7";
NETWORK
TITLE = BACKWARD
      A(;
      O     "M 78.5";
      O     "M 78.6";
      );
      L     S5T#500MS;
      SF    "T101";
      NOP   0;
      NOP   0;
      NOP   0;
      A     "T101";
      =     "A 9.3";
NETWORK
TITLE = CONVEYOR BRAKE
      A(;
      O     "M 78.5";
      O     "M 78.6";
      );
      A     "AUTO";
      L     S5T#20S;
      SD    "T102";
NETWORK
TITLE = RUNTIME MONITORING
      A     "T102";
      =     "M 78.7";
END_FUNCTION

FUNCTION "CONVEYOR_6" : VOID	// FC 76
TITLE = CONVEYOR POS.6
//
//Bits for conveyor control:
//Bit 0 = Locking conveyor
//Bit 1 = Spare
//Bit 2 = Run in
//Bit 3 = Occupied
//Bit 4 = Run out
//Bit 5 = Forward
//Bit 6 = Backward
//Bit 7 = Runtime
VERSION : 0.1
BEGIN
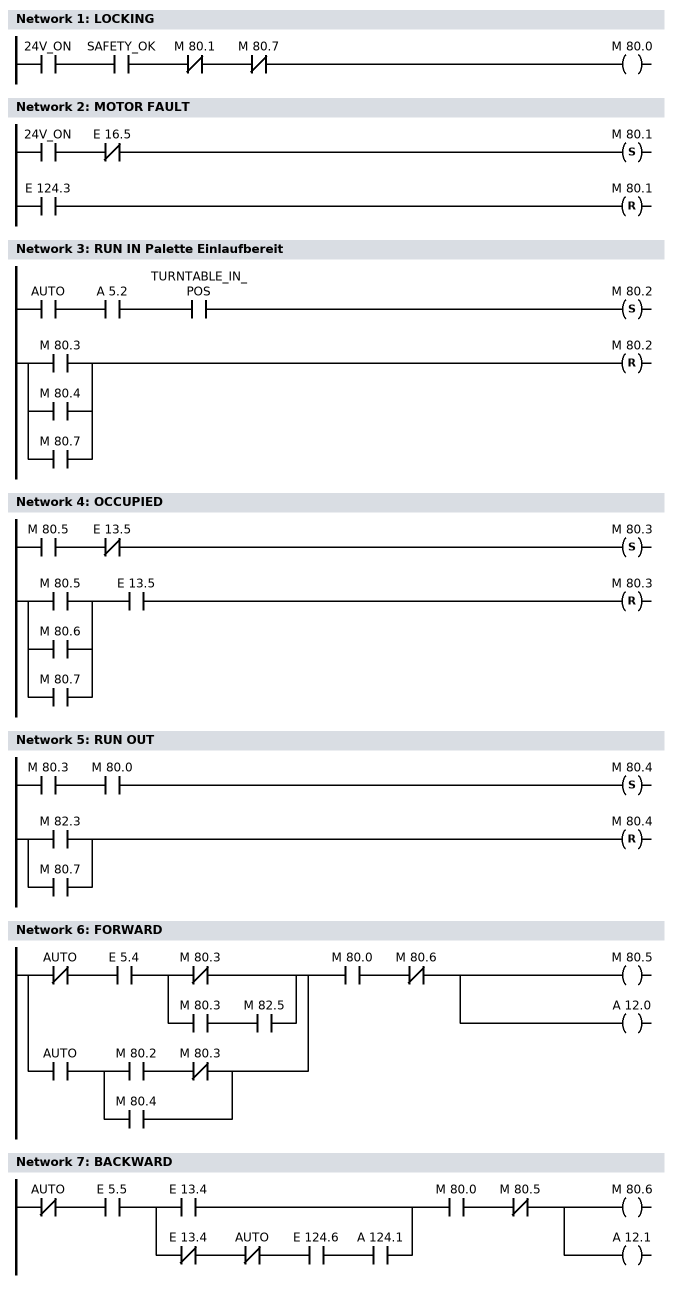
NETWORK
TITLE = LOCKING
      A     "24V_ON";
      A     "SAFETY_OK";
      AN    "M 80.1";
      AN    "M 80.7";
      =     "M 80.0";
NETWORK
TITLE = MOTOR FAULT
      A     "24V_ON";
      AN    "E 16.5";
      S     "M 80.1";
      A     "E 124.3";
      R     "M 80.1";
      NOP   0;
NETWORK
TITLE = RUN IN Palette Einlaufbereit
      A     "AUTO";
      A     "A 5.2";
      A     "TURNTABLE_IN_POS";
      S     "M 80.2";
      A(;
      O     "M 80.3";
      O     "M 80.4";
      O     "M 80.7";
      );
      R     "M 80.2";
      NOP   0;
NETWORK
TITLE = OCCUPIED
      A     "M 80.5";
      AN    "E 13.5";
      S     "M 80.3";
      A(;
      O     "M 80.5";
      O     "M 80.6";
      O     "M 80.7";
      );
      A     "E 13.5";
      R     "M 80.3";
      NOP   0;
NETWORK
TITLE = RUN OUT
      A     "M 80.3";
      A     "M 80.0";
      S     "M 80.4";
      A(;
      O     "M 82.3";
      O     "M 80.7";
      );
      R     "M 80.4";
      NOP   0;
NETWORK
TITLE = FORWARD
      A(;
      AN    "AUTO";
      A     "E 5.4";
      A(;
      ON    "M 80.3";
      O;
      A     "M 80.3";
      A     "M 82.5";
      );
      O;
      A     "AUTO";
      A(;
      A     "M 80.2";
      AN    "M 80.3";
      O     "M 80.4";
      );
      );
      A     "M 80.0";
      AN    "M 80.6";
      =     "M 80.5";
      =     "A 12.0";
NETWORK
TITLE = BACKWARD
      AN    "AUTO";
      A     "E 5.5";
      A(;
      O     "E 13.4";
      O;
      AN    "E 13.4";
      AN    "AUTO";
      A     "E 124.6";
      A     "A 124.1";
      );
      A     "M 80.0";
      AN    "M 80.5";
      =     "M 80.6";
      =     "A 12.1";
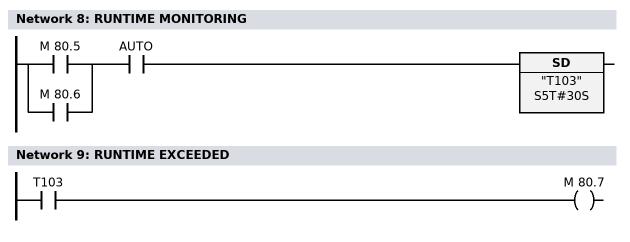
NETWORK
TITLE = RUNTIME MONITORING
      A(;
      O     "M 80.5";
      O     "M 80.6";
      );
      A     "AUTO";
      L     S5T#30S;
      SD    "T103";
NETWORK
TITLE = RUNTIME EXCEEDED
      A     "T103";
      =     "M 80.7";
END_FUNCTION

FUNCTION "CONVEYOR_7" : VOID	// FC 77
TITLE = CONVEYOR POS.7
//
//Bits for conveyor control:
//Bit 0 = Locking conveyor
//Bit 1 = Spare
//Bit 2 = Run in
//Bit 3 = Occupied
//Bit 4 = Run out
//Bit 5 = Forward
//Bit 6 = Backward
//Bit 7 = Runtime
VERSION : 0.1
BEGIN
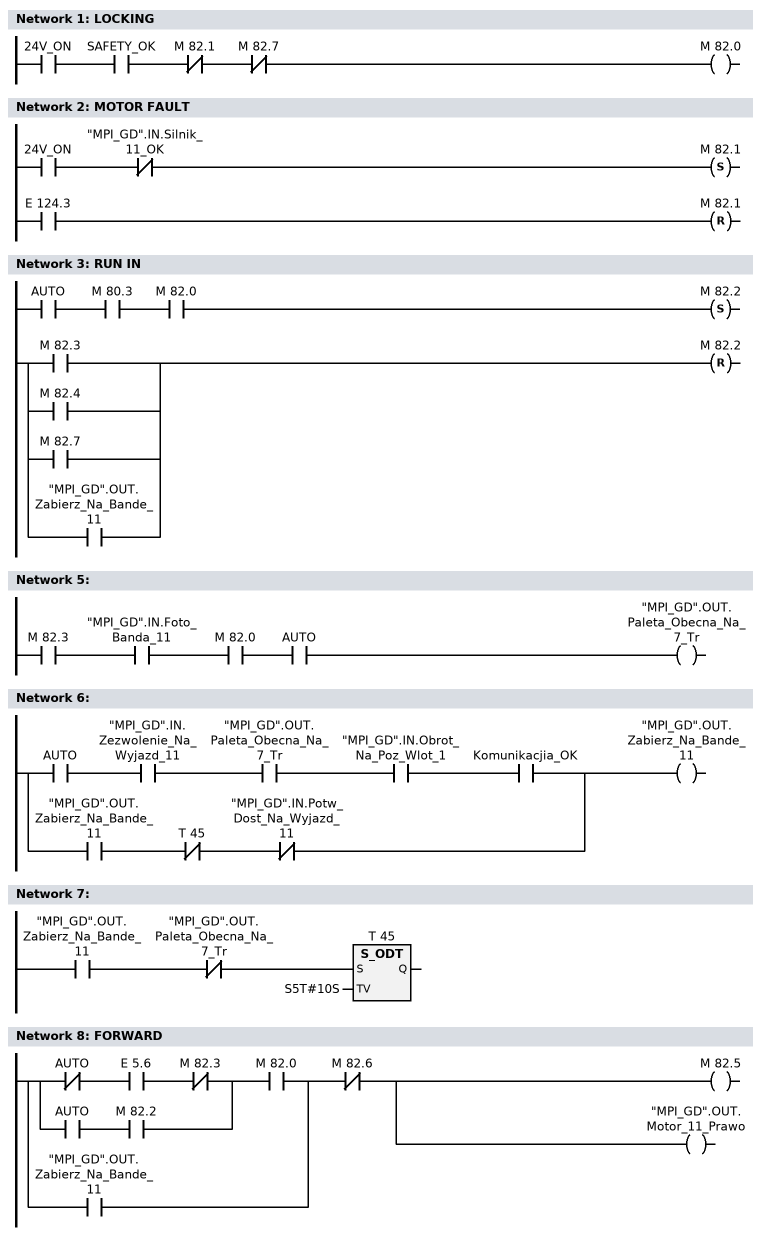
NETWORK
TITLE = LOCKING
      A     "24V_ON";
      A     "SAFETY_OK";
      AN    "M 82.1";
      AN    "M 82.7";
      =     "M 82.0";
NETWORK
TITLE = MOTOR FAULT
      A     "24V_ON";
      AN    "MPI_GD".IN.Silnik_11_OK;
      S     "M 82.1";
      A     "E 124.3";
      R     "M 82.1";
      NOP   0;
NETWORK
TITLE = RUN IN
//Wjazd na przenosnik 7
      A     "AUTO";
      A     "M 80.3";
      A     "M 82.0";
      S     "M 82.2";
      A(;
      O     "M 82.3";
      O     "M 82.4";
      O     "M 82.7";
      O     "MPI_GD".OUT.Zabierz_Na_Bande_11;
      );
      R     "M 82.2";
      NOP   0;
NETWORK
TITLE = OCCUPIED
//Tasma zajeta
      A(;
      A     "MPI_GD".IN.Foto_Banda_11;
      S     "M 82.3";
      A(;
      O     "M 82.6";
      O     "M 82.7";
      O;
      AN    "MPI_GD".OUT.Zabierz_Na_Bande_11;
      AN    T 46;
      );
      AN    "MPI_GD".IN.Foto_Banda_11;
      R     "M 82.3";
      A     "M 82.3";
      );
      A     "MPI_GD".IN.Foto_Banda_11;
      L     S5T#12S;
      SF    T 46;
NETWORK
TITLE =
      A     "M 82.3";
      A     "MPI_GD".IN.Foto_Banda_11;
      A     "M 82.0";
      A     "AUTO";
      =     "MPI_GD".OUT.Paleta_Obecna_Na_7_Tr;
NETWORK
TITLE =
//Spelnienie warunkow na wjazd na obrotnice
      A     "AUTO";
      A     "MPI_GD".IN.Zezwolenie_Na_Wyjazd_11;
      A     "MPI_GD".OUT.Paleta_Obecna_Na_7_Tr;
      A     "MPI_GD".IN.Obrot_Na_Poz_Wlot_1;
      A     "Komunikacjia_OK";
      O;
      A     "MPI_GD".OUT.Zabierz_Na_Bande_11;
      AN    T 45;
      AN    "MPI_GD".IN.Potw_Dost_Na_Wyjazd_11;
      =     "MPI_GD".OUT.Zabierz_Na_Bande_11;
NETWORK
TITLE =
//Czas kontrolny
      A     "MPI_GD".OUT.Zabierz_Na_Bande_11;
      AN    "MPI_GD".OUT.Paleta_Obecna_Na_7_Tr;
      L     S5T#10S;
      SD    T 45;
      NOP   0;
      NOP   0;
      NOP   0;
      NOP   0;
NETWORK
TITLE = FORWARD
//Bylo q12.2
      A(;
      A(;
      AN    "AUTO";
      A     "E 5.6";
      AN    "M 82.3";
      O;
      A     "AUTO";
      A     "M 82.2";
      );
      A     "M 82.0";
      O     "MPI_GD".OUT.Zabierz_Na_Bande_11;
      );
      AN    "M 82.6";
      =     "M 82.5";
      =     "MPI_GD".OUT.Motor_11_Prawo;
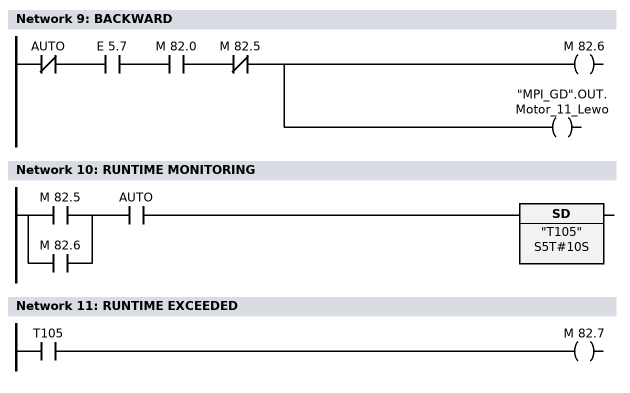
NETWORK
TITLE = BACKWARD
//bylo q12.3
      AN    "AUTO";
      A     "E 5.7";
      A     "M 82.0";
      AN    "M 82.5";
      =     "M 82.6";
      =     "MPI_GD".OUT.Motor_11_Lewo;
NETWORK
TITLE = RUNTIME MONITORING
      A(;
      O     "M 82.5";
      O     "M 82.6";
      );
      A     "AUTO";
      L     S5T#10S;
      SD    "T105";
NETWORK
TITLE = RUNTIME EXCEEDED
      A     "T105";
      =     "M 82.7";
END_FUNCTION

FUNCTION "CONV_2" : VOID	// FC 92
VERSION : 0.1
BEGIN
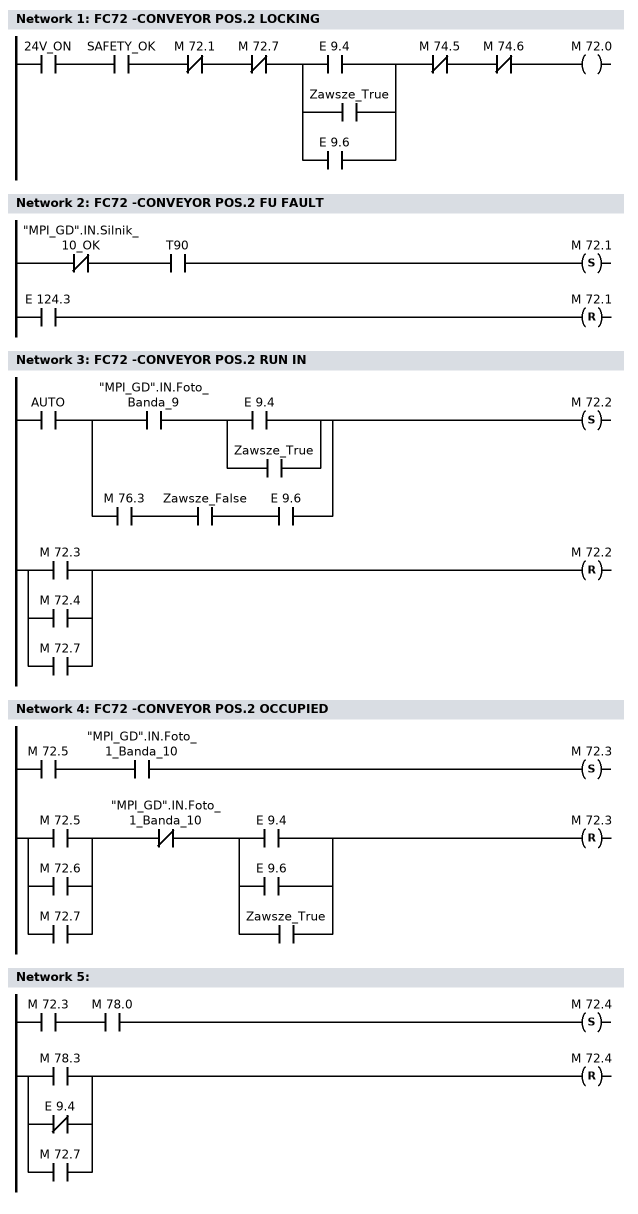
NETWORK
TITLE = FC72 -CONVEYOR POS.2 LOCKING
//Ustawienie obrotnicy na pozycji 0 stopni
      A     "24V_ON";
      A     "SAFETY_OK";
      AN    "M 72.1";
      AN    "M 72.7";
      A(;
      O     "E 9.4";
      O     "Zawsze_True";
      O     "E 9.6";
      );
      AN    "M 74.5";
      AN    "M 74.6";
      =     "M 72.0";
NETWORK
TITLE = FC72 -CONVEYOR POS.2 FU FAULT
//Silnik przenosnika jest OK
      AN    "MPI_GD".IN.Silnik_10_OK;
      A     "T90";
      S     "M 72.1";
      A     "E 124.3";
      R     "M 72.1";
      NOP   0;
NETWORK
TITLE = FC72 -CONVEYOR POS.2 RUN IN
//Wjazd palet na bande
      A     "AUTO";
      A(;
      A     "MPI_GD".IN.Foto_Banda_9;
      A(;
      O     "E 9.4";
      O     "Zawsze_True";
      );
      O;
      A     "M 76.3";
      A     "Zawsze_False";
      A     "E 9.6";
      );
      S     "M 72.2";
      A(;
      O     "M 72.3";
      O     "M 72.4";
      O     "M 72.7";
      );
      R     "M 72.2";
      NOP   0;
NETWORK
TITLE = FC72 -CONVEYOR POS.2 OCCUPIED
//Paleta na przenosniku nr 2 
      A     "M 72.5";
      A     "MPI_GD".IN.Foto_1_Banda_10;
      S     "M 72.3";
      A(;
      O     "M 72.5";
      O     "M 72.6";
      O     "M 72.7";
      );
      AN    "MPI_GD".IN.Foto_1_Banda_10;
      A(;
      O     "E 9.4";
      O     "E 9.6";
      O     "Zawsze_True";
      );
      R     "M 72.3";
      NOP   0;
NETWORK
TITLE =
      A     "M 72.3";
      A     "M 78.0";
      S     "M 72.4";
      A(;
      O     "M 78.3";
      ON    "E 9.4";
      O     "M 72.7";
      );
      R     "M 72.4";
      NOP   0;
